SUBAPPLICATION Uebung_103c2 (* DigitalInput_I1 auf DigitalOutput_Q1, mit Plug and Socket und DEMUX *)
  (* Standard: 61499-2; Description: Copyright (c) 2023 Meisterschulen am Ostbahnhof This program and the accompanying materials are made available under the terms of the Eclipse Public License 2.0 which is available at https://www.eclipse.org/legal/epl-2.0/ SPDX-License-Identifier: EPL-2.0 *)
  (* Version 1.0, 2023-10-23, Franz Höpfinger, Meisterschulen am Ostbahnhof *)
  PACKAGE Uebungen;
  IMPORT logiBUS::io::DI::logiBUS_DI::Input_I1;
  IMPORT logiBUS::io::DQ::logiBUS_DO::Output_Q1;
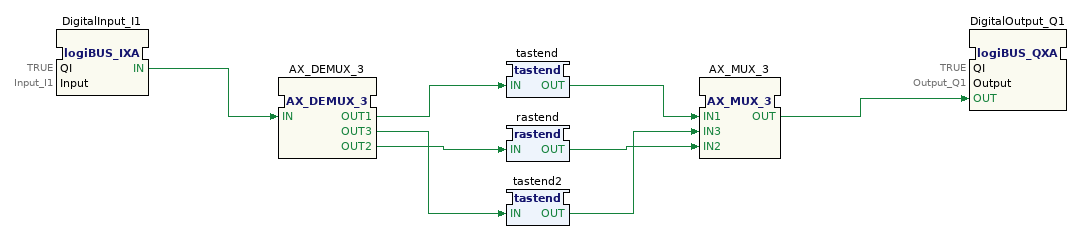
  FBS
    DigitalInput_I1 : logiBUS::io::DI::logiBUS_IXA(QI := TRUE, Input := Input_I1);
    DigitalOutput_Q1 : logiBUS::io::DQ::logiBUS_QXA(QI := TRUE, Output := Output_Q1);
    AX_DEMUX_3 : adapter::selection::unidirectional::AX_DEMUX_3;
    AX_MUX_3 : adapter::selection::unidirectional::AX_MUX_3;
  END_FBS
  SUBAPPS
    rastend : MyLib::sys::rastend;
    tastend : MyLib::sys::tastend;
    tastend2 : MyLib::sys::tastend;
  END_SUBAPPS
  ADAPTER_CONNECTIONS
    AX_MUX_3.OUT TO DigitalOutput_Q1.OUT;
    DigitalInput_I1.IN TO AX_DEMUX_3.IN;
    AX_DEMUX_3.OUT1 TO tastend.IN;
    tastend.OUT TO AX_MUX_3.IN1;
    AX_DEMUX_3.OUT3 TO tastend2.IN;
    tastend2.OUT TO AX_MUX_3.IN3;
    rastend.OUT TO AX_MUX_3.IN2;
    AX_DEMUX_3.OUT2 TO rastend.IN;
  END_CONNECTIONS
END_SUBAPPLICATION
